// TIA Portal V19 export
ORGANIZATION_BLOCK "Startup"   // OB2103, LAD, Startup
TITLE = "Complete Restart"
// stored: AutoNumber false, IsIECCheckEnabled true, Namespace Unit2.EM0, SetENOAutomatically true
   VAR_INPUT
      LostRetentive : Bool;   // True if retentive data are lost
      LostRTC : Bool;   // True if date and time are lost
   END_VAR
BEGIN

REGION Network 1 (SCL): Build the Absolut Reference Designator
   // Set the Absoult Reference Designator in the Config DB
   IF LEN(IN := "Unit2.EM0.Config".em.referenceDesignator.parent) <> 0 THEN
       "Unit2.EM0.Config".em.referenceDesignator.combined := CONCAT_WSTRING(IN1 := "Unit2.EM0.Config".em.referenceDesignator.parent, IN2 := WSTRING#'.', IN3 := "Unit2.EM0.Config".em.referenceDesignator.relative);
   ELSE
       "Unit2.EM0.Config".em.referenceDesignator.combined := "Unit2.EM0.Config".em.referenceDesignator.relative;
   END_IF;
END_REGION

REGION Network 2 (SCL): Assign axes data
   // This is an example how to assign axes to DB_ANY in DB Config. If you have axes, assign them here. The Config.axis[] variables will be handed over to the control modules. That enables a flexible programming.
   // // Assign axes
   // Config.axis[1] := PositioningAxis;
   // Config.axis[2] := SynchronousAxis;
END_REGION
END_ORGANIZATION_BLOCK
